// TIA Portal V20 export
TYPE "AnalogOutput_DT"
   STRUCT
      SWRealValue : Real;   // Software real value use in PLC
      HWWordValue : Word;   // Hardware value direclty to physical input
   END_STRUCT;
END_TYPE
